Staubli VAL3: onF8Event.pgx

program onF8Event()
begin
   // look if the bButton is enable
  if bButton[7]
    //
  endIf
end
